// TIA Portal V21 export
TYPE "Rcp_V100_Type"
   STRUCT
      RecipeName { S7_SetPoint := 'True'} : "Rcp_Name_Type";
      General { S7_SetPoint := 'True'} : "Rcp_Generale";
      Filler { S7_SetPoint := 'True'} : "Rcp_Filler";
      VacuumFiller { S7_SetPoint := 'True'} : "Rcp_VacuumFiller";
      Capper { S7_SetPoint := 'True'} : "Rcp_Capper";
      "Blower / Rinser" { S7_SetPoint := 'True'} : "Rcp_Blower&Rinser";
   END_STRUCT;
END_TYPE
